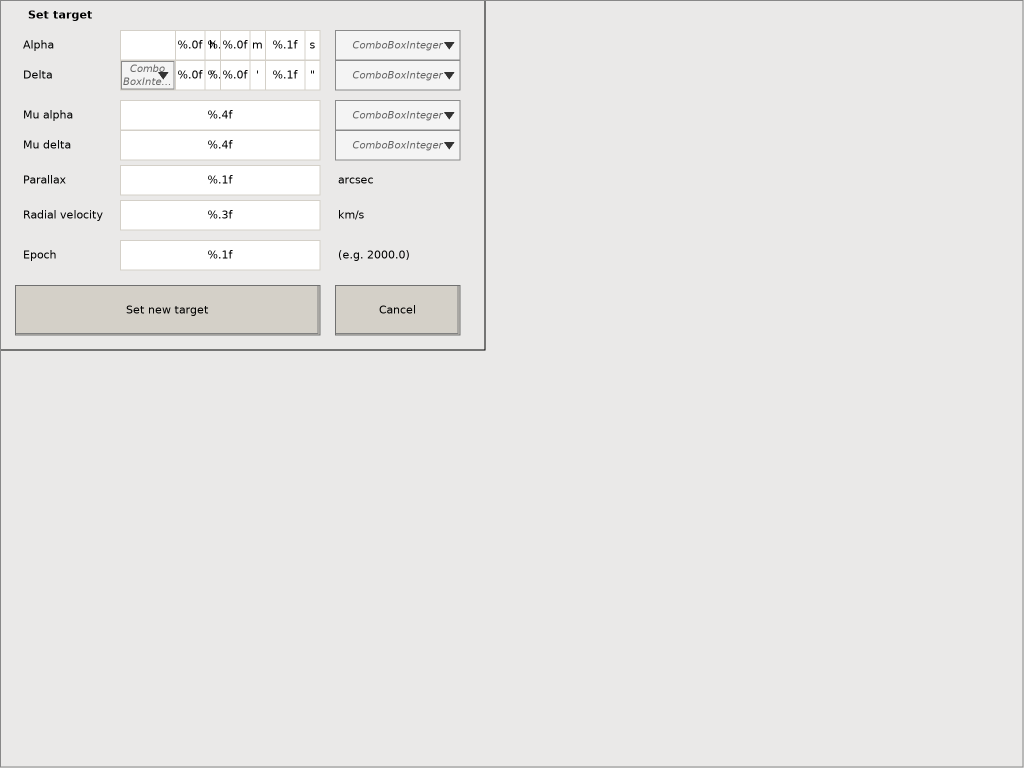
VISUALIZATION VISU_AxesSetTargetDialog  // 1024x768
    Rectangle (0,0 485x350)
    Label (25,5 95x20), "Set target"
    Label (20,30 95x30), "Alpha"
    Label (20,60 95x30), "Delta"
    Textfield (120,30 200x30), "%.8f", text variable: GLOBAL.gui.axes.setTarget.field_alpha_decimal, invisible if: GLOBAL.gui.axes.setTarget.units_alpha = AxesDialogAlphaUnits.DIALOG_HMS
        OnMouseClick: write the text variable via VisuDialogs.Numpad
    Textfield (120,60 200x30), "%.8f", text variable: GLOBAL.gui.axes.setTarget.field_delta_decimal, invisible if: GLOBAL.gui.axes.setTarget.units_delta = AxesDialogDeltaUnits.DIALOG_DMS
        OnMouseClick: write the text variable via VisuDialogs.Numpad
    Label (20,100 95x30), "Mu alpha"
    Label (20,130 95x30), "Mu delta"
    Textfield (120,100 200x30), "%.4f", text variable: GLOBAL.gui.axes.setTarget.field_muAlpha
        OnMouseClick: write the text variable via VisuDialogs.Numpad
    Label (20,165 95x30), "Parallax"
    Label (20,200 95x30), "Radial velocity"
    Label (335,200 80x30), "km/s"
    Label (335,165 80x30), "arcsec"
    Textfield (120,130 200x30), "%.4f", text variable: GLOBAL.gui.axes.setTarget.field_muDelta
        OnMouseClick: write the text variable via VisuDialogs.Numpad
    Textfield (120,165 200x30), "%.1f", text variable: GLOBAL.gui.axes.setTarget.field_parallax
        OnMouseClick: write the text variable via VisuDialogs.Numpad
    Textfield (120,200 200x30), "%.3f", text variable: GLOBAL.gui.axes.setTarget.field_radialVelocity
        OnMouseClick: write the text variable via VisuDialogs.Numpad
    Label (20,240 95x30), "Epoch"
    Label (335,240 80x30), "(e.g. 2000.0)"
    Textfield (120,240 200x30), "%.1f", text variable: GLOBAL.gui.axes.setTarget.field_epoch
        OnMouseClick: write the text variable via VisuDialogs.Numpad
    Button (15,285 305x50), "Set new target", input disabled if: GLOBAL.mtcs.parts.axes.processes.setTarget.statuses.enabledStatus.disabled
        OnMouseClick: execute { GLOBAL.gui.axes.setTarget.do_request := TRUE; }
        OnMouseClick: CloseDialog Dialog=VISU_AxesPointDialog, Result=OK, NumpadKeypadSet=True
    ComboBoxInteger (335,30 125x30), variable: GLOBAL.gui.axes.setTarget.units_alpha, text list: 'AxesDialogAlphaUnitsTextList'
    ComboBoxInteger (335,60 125x30), variable: GLOBAL.gui.axes.setTarget.units_delta, text list: 'AxesDialogDeltaUnitsTextList'
    ComboBoxInteger (335,100 125x30), variable: GLOBAL.gui.axes.setTarget.units_mu, text list: 'AxesMuUnitsTextList'
    Button (335,285 125x50), "Cancel"
        OnMouseClick: CloseDialog Dialog=VISU_AxesSetTargetDialog, Result=Cancel, NumpadKeypadSet=True
    ComboBoxInteger (335,130 125x30), variable: GLOBAL.gui.axes.setTarget.units_mu, text list: 'AxesMuUnitsTextList'
    Textfield (175,60 30x30), "%.0f", text variable: GLOBAL.gui.axes.setTarget.field_delta_d, invisible if: GLOBAL.gui.axes.setTarget.units_delta <> AxesDialogDeltaUnits.DIALOG_DMS
        OnMouseClick: write the text variable via VisuDialogs.Numpad
    ComboBoxInteger (121,61 53x28), variable: GLOBAL.gui.axes.setTarget.field_delta_sign, invisible if: GLOBAL.gui.axes.setTarget.units_delta <> AxesDialogDeltaUnits.DIALOG_DMS, text list: 'AxesDialogSignTextList'
    Textfield (220,60 30x30), "%.0f", text variable: GLOBAL.gui.axes.setTarget.field_delta_m, invisible if: GLOBAL.gui.axes.setTarget.units_delta <> AxesDialogDeltaUnits.DIALOG_DMS
        OnMouseClick: write the text variable via VisuDialogs.Numpad
    Textfield (265,60 40x30), "%.1f", text variable: GLOBAL.gui.axes.setTarget.field_delta_s, invisible if: GLOBAL.gui.axes.setTarget.units_delta <> AxesDialogDeltaUnits.DIALOG_DMS
        OnMouseClick: write the text variable via VisuDialogs.Numpad
    Label (205,60 15x30), "°", invisible if: GLOBAL.gui.axes.setTarget.units_delta <> AxesDialogDeltaUnits.DIALOG_DMS
    Label (250,60 15x30), "'", invisible if: GLOBAL.gui.axes.setTarget.units_delta <> AxesDialogDeltaUnits.DIALOG_DMS
    Label (305,60 15x30), """, invisible if: GLOBAL.gui.axes.setTarget.units_delta <> AxesDialogDeltaUnits.DIALOG_DMS
    Textfield (175,30 30x30), "%.0f", text variable: GLOBAL.gui.axes.setTarget.field_alpha_h, invisible if: GLOBAL.gui.axes.setTarget.units_alpha <> AxesDialogAlphaUnits.DIALOG_HMS
        OnMouseClick: write the text variable via VisuDialogs.Numpad
    Textfield (220,30 30x30), "%.0f", text variable: GLOBAL.gui.axes.setTarget.field_alpha_m, invisible if: GLOBAL.gui.axes.setTarget.units_alpha <> AxesDialogAlphaUnits.DIALOG_HMS
        OnMouseClick: write the text variable via VisuDialogs.Numpad
    Textfield (265,30 40x30), "%.1f", text variable: GLOBAL.gui.axes.setTarget.field_alpha_s, invisible if: GLOBAL.gui.axes.setTarget.units_alpha <> AxesDialogAlphaUnits.DIALOG_HMS
        OnMouseClick: write the text variable via VisuDialogs.Numpad
    Label (205,30 15x30), "h", invisible if: GLOBAL.gui.axes.setTarget.units_alpha <> AxesDialogAlphaUnits.DIALOG_HMS
    Label (250,30 15x30), "m", invisible if: GLOBAL.gui.axes.setTarget.units_alpha <> AxesDialogAlphaUnits.DIALOG_HMS
    Label (305,30 15x30), "s", invisible if: GLOBAL.gui.axes.setTarget.units_alpha <> AxesDialogAlphaUnits.DIALOG_HMS
END_VISUALIZATION

(* stored: Version 1.1.0.1, ProductVersion 3.1.4019.2
   Visu VISU_AxesSetTargetDialog: Id {e5235c55-e427-4098-b845-3e1564bdbc81} *)
